FUNCTION Camera_Update : Camera_Error
VAR_IN_OUT
	Camera : Cognex_Camera;
END_VAR

IF Camera.CameraState = Camera_State.Idel THEN
	RETURN;
ELSIF Camera.CameraState = Camera_State.Jope_Running THEN
	Update_Jobe_State(Camera);
ELSIF Camera.CameraState = Camera_State.Command_Running THEN
	Update_Jobe_State(Camera);
ELSIF Camera.CameraState = Camera_State.Clear_Error THEN
	Camera.Inspection.Clear_Error := FALSE;
	Camera.CameraState := Camera_State.Idel;
ELSE
	Camera_Update := Camera.Error;
END_IF

END_FUNCTION

(* stored: Version 1.1.0.1, ProductVersion 3.1.4024.10
   POU Camera_Update: Id {85bb63c0-efb5-40a9-b294-e539bdfb8a90}, SpecialFunc None *)
